FUNCTION_BLOCK Brake
VAR_INPUT
	Lh_off:BOOL;(*Left brake off signal - usually from left spring nest*)
	Lh_rubbing:BOOL; (*Left brake rubbing signal - usually from left spring nest*)
	Lh_on:BOOL; (*Left brake on signal - usually from left spring nest*)
	Lh_wear:BOOL; (*Left brake wear signal - usually from left spring nest*)
	Rh_off:BOOL; (*Right brake on signal - usually from right spring nest*)
	Rh_rubbing:BOOL; (*Right brake rubbing signal - usually from right spring nest*)
	Rh_on:BOOL; (*Right brake on signal - usually from right spring nest*)
	Rh_wear:BOOL; (*Right brake wear signal - usually from Right spring nest*)
	Lever_on:BOOL; (*Brake lever on limit switch*)
	Lever_off:BOOL; (*Brake lever off - normally from same limit switch as "Lever_on"*)
	Lever_fully_off:BOOL; (*Brake lever fully off limit switch. Necessary for automatic winders.*)
	Lh_test:BOOL; (*Left brake test switch - normally on driver's desk. Often the same switch as Lh_dump.*)
	Rh_test:BOOL; (*Right brake test switch - normally on driver's desk. Often the same switch as Rh_dump.*)
	Lh_dump:BOOL; (*Left brake dump switch - normally on driver's desk. Often the same switch as Lh_test.*)
	Rh_dump:BOOL; (*Right brake dump switch - normally on driver's desk. Often the same switch as Rh_test.*)
	Maintenance_switch:BOOL; (*Brake maintenance switch (can be on driver's desk or in control panels).*)
	Trail_brakes:BOOL; (*Trail brake control signal. Used to disable Lh_not_fully_off and Rh_not_fully_off trips.*)
	Lh_speed:INT; (*Left drum speed (normally in mm/s)*)
	Rh_speed:INT; (*Right drum speed (normally in mm/s)*)
	Movement_detect:BOOL; (*Drum movement detected (on either of the two drums in a double-drum winder)*)
	On_time:TIME; (*Maximum time allowed for brakes to apply.*)
	Off_time:TIME; (*Maximum time allowed for brakes to lift.*)
	Rubbing_speed:INT; (*Speed above which the brakes must be above the rubbing position*)
	Rubbing_time:TIME; (*Time before brake rubbing trips trigger *)
END_VAR
VAR_OUTPUT
	Maintenance:BOOL; (*The winder is in brake maintenance mode*)
	Proved_on:BOOL; (*The brake lever (if in manual mode) and both brakes are on*)
	Proved_on_500ms:BOOL; (*The brakes have been proved on for 500ms*)
	cs_Lh_off_before_rubbing:BOOL; (*The Lh_off switch has closed but the Lh_rubbing switch has not yet closed*)
	cs_Lh_on_and_rubbing:BOOL; (*The Lh_on switch has closed but the Lh_rubbing switch is still closed*)
	cs_Lh_wear_before_on:BOOL; (*The Lh_on switch has closed but the Lh_rubbing switch is still closed*)
	cs_Lh_on_and_off:BOOL; (*The Lh_on and Lh_off switches are simultaneously closed*)
	cs_Rh_off_before_rubbing:BOOL; (*The Rh_off switch has closed but the Rh_rubbing switch has not yet closed*)
	cs_Rh_on_and_rubbing:BOOL; (*The Rh_on switch has closed but the Rh_rubbing switch is still closed*)
	cs_Rh_wear_before_on:BOOL; (*The Rh_on switch has closed but the Rh_rubbing switch is still closed*)
	cs_Rh_on_and_off:BOOL; (*The Rh_on and Rh_off switches are simultaneously closed*)
	cs_Lever_off_and_on:BOOL; (*The brake lever on and off switches are simultaneously closed*)
	cs_Lever_fully_off_and_on:BOOL; (*The brake lever on and fully off switches are simultaneously closed*)
	cs_Lh_not_fully_off:BOOL; (*The brake lever has been off for longer than the brake lift time but the Lh_off switch is not closed. Trail_brakes disables this fault.*)
	cs_Rh_not_fully_off:BOOL; (*The brake lever has been off for longer than the brake lift time but the Rh_off switch is not closed. Trail_brakes disables this fault.*)
	tr_Lh_not_on:BOOL; (*The brake lever has been on for longer than the brake application time but the Lh_on switch is not closed.*)
	tr_Rh_not_on:BOOL; (*The brake lever has been on for longer than the brake application time but the Rh_on switch is not closed.*)
	tr_Lh_rubbing_trip:BOOL; (*Lh_rubbing active above the rubbing trip speed*)
	tr_Rh_rubbing_trip:BOOL; (*Rh_rubbing active above the rubbing trip speed*)
	tr_No_brake_on_in_maint:BOOL; (*The power lever was moved from the neutral position in brake maintenance mode*)
	tr_Movement_in_maint:BOOL; (*Movement has been detected in brake maintenance mode*)
	tr_Maint_switch_on:BOOL; (*The brake maintenance switch is on but a brake is not dumped*)
	hmi_Status:ARRAY[1..2] OF WORD; (*Status bits for HMI*)
END_VAR
VAR
	TON_0: TON;
	Maintenance_req: BOOL;
	RS_0: RS;
	TON_1: TON;
	TON_2: TON;
	TON_3: TON;
	TON_4: TON;
	TON_5: TON;
	TON_6: TON;
	TON_7: TON;
	TON_8: TON;
	TON_9: TON;
	TON_10: TON;
	TON_11: TON;
	TON_12: TON;
	TON_13: TON;
	TON_14: TON;
	TON_15: TON;
	TON_16: TON;
	TON_17: TON;
	BIT_TO_WORD_V0_0: BIT_TO_WORD_V0;
	BIT_TO_WORD_V0_1: BIT_TO_WORD_V0;
END_VAR

Brake_data_m();
Brake_faults();

METHOD Brake_data_m
VAR_INPUT
END_VAR
VAR
END_VAR
VAR_INST // added by the converter: edge detectors and wires of the graphical bodies
    _w1, _w2, _w3, _w4 : BOOL;
END_VAR
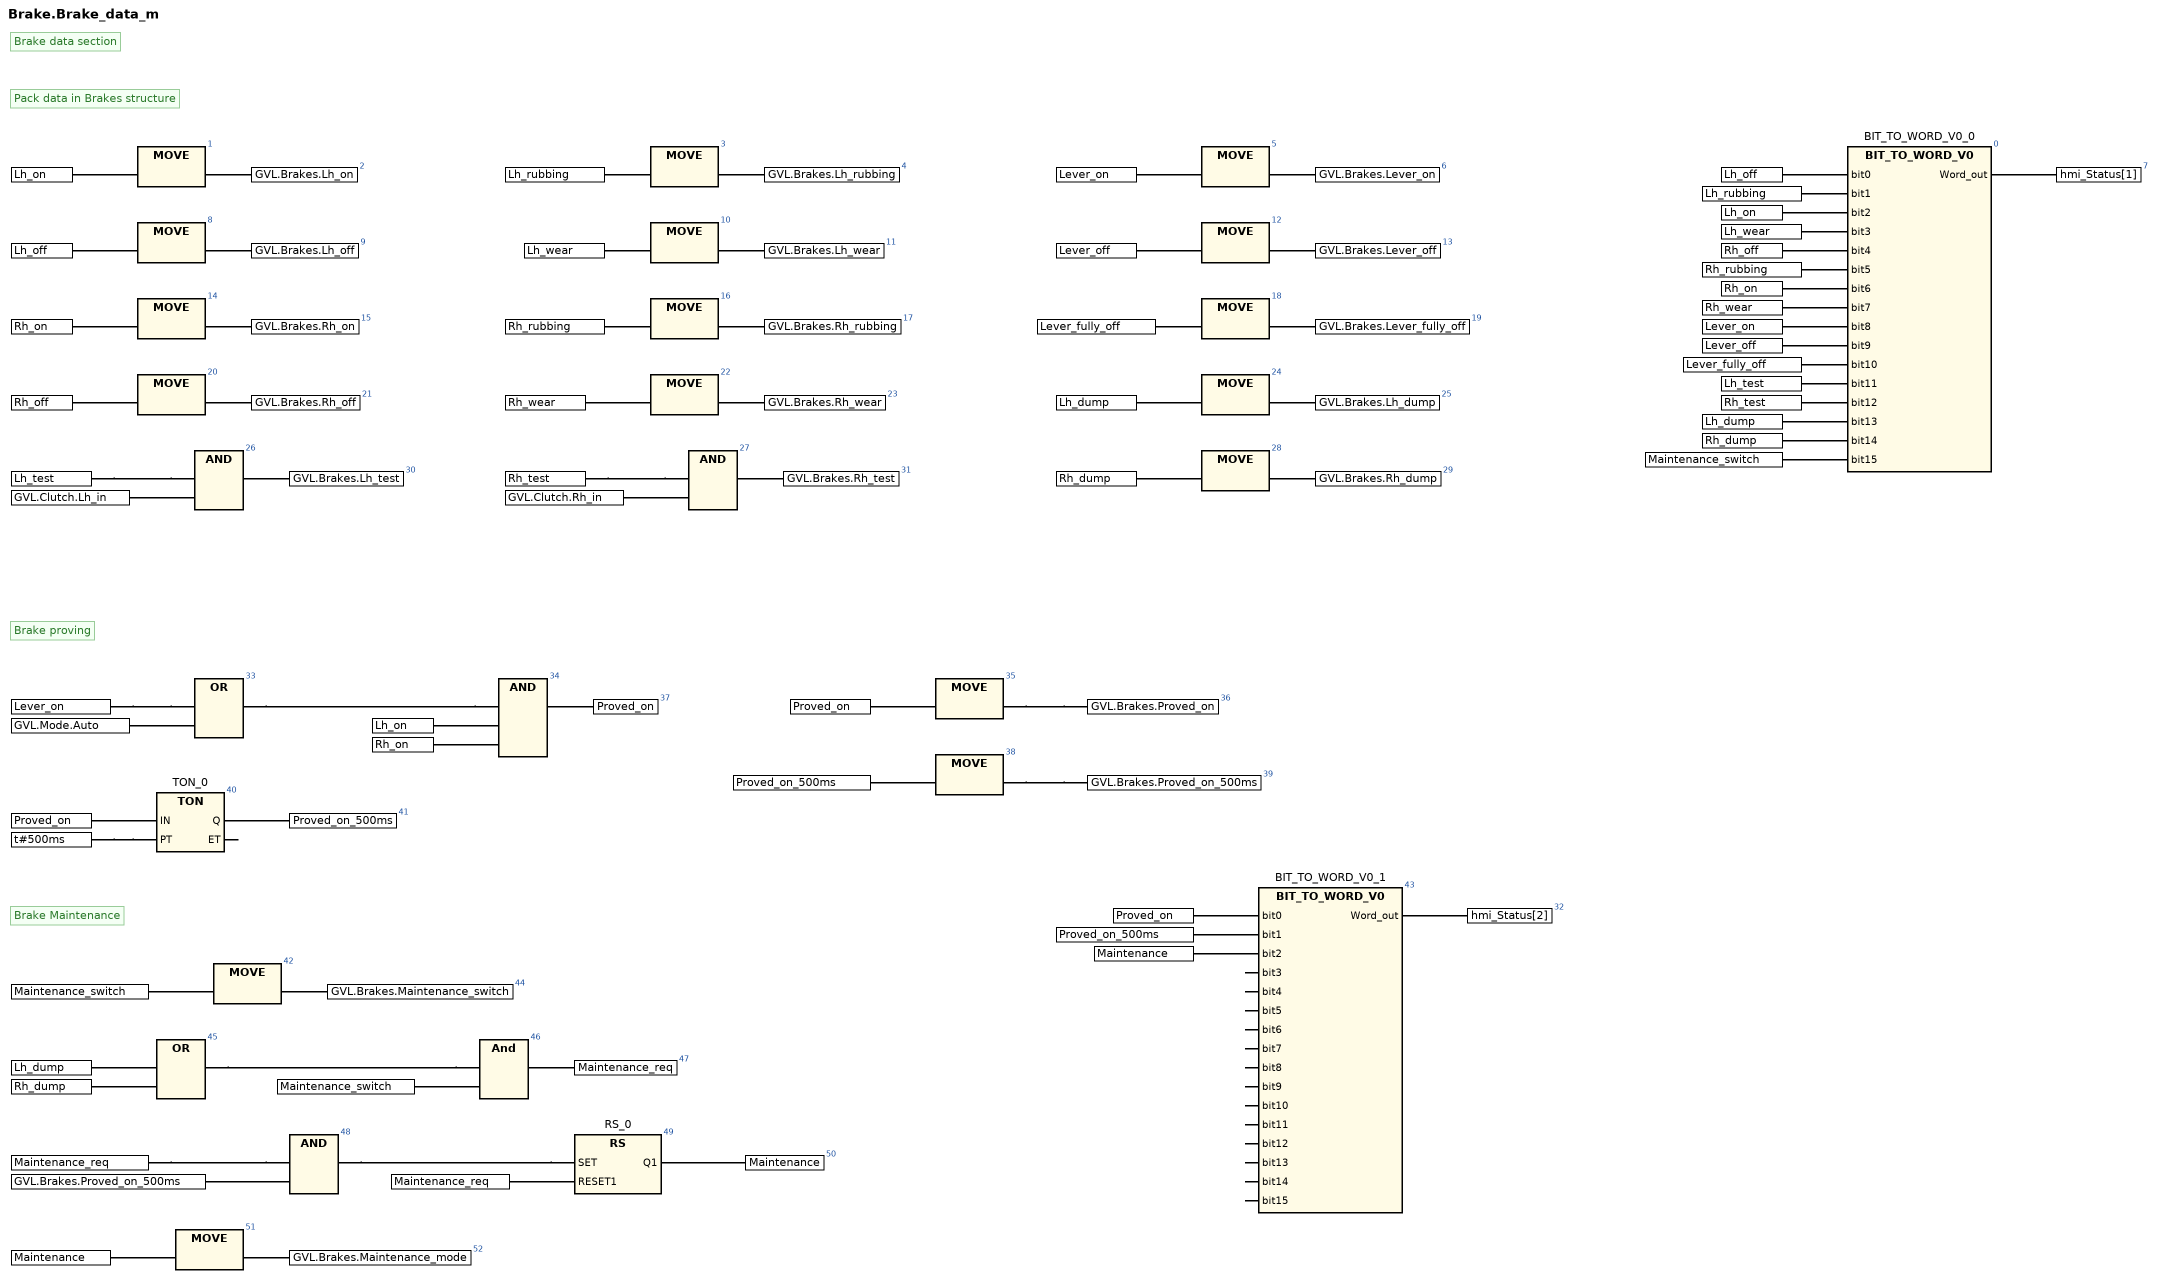
BIT_TO_WORD_V0_0(
    bit0 := Lh_off,
    bit1 := Lh_rubbing,
    bit2 := Lh_on,
    bit3 := Lh_wear,
    bit4 := Rh_off,
    bit5 := Rh_rubbing,
    bit6 := Rh_on,
    bit7 := Rh_wear,
    bit8 := Lever_on,
    bit9 := Lever_off,
    bit10 := Lever_fully_off,
    bit11 := Lh_test,
    bit12 := Rh_test,
    bit13 := Lh_dump,
    bit14 := Rh_dump,
    bit15 := Maintenance_switch); // BIT_TO_WORD_V0
// Brake data section
// Pack data in Brakes structure
GVL.Brakes.Lh_on := Lh_on;
GVL.Brakes.Lh_rubbing := Lh_rubbing;
GVL.Brakes.Lever_on := Lever_on;
hmi_Status[1] := BIT_TO_WORD_V0_0.Word_out;
GVL.Brakes.Lh_off := Lh_off;
GVL.Brakes.Lh_wear := Lh_wear;
GVL.Brakes.Lever_off := Lever_off;
GVL.Brakes.Rh_on := Rh_on;
GVL.Brakes.Rh_rubbing := Rh_rubbing;
GVL.Brakes.Lever_fully_off := Lever_fully_off;
GVL.Brakes.Rh_off := Rh_off;
GVL.Brakes.Rh_wear := Rh_wear;
GVL.Brakes.Lh_dump := Lh_dump;
_w1 := Lh_test AND GVL.Clutch.Lh_in;
_w2 := Rh_test AND GVL.Clutch.Rh_in;
GVL.Brakes.Rh_dump := Rh_dump;
GVL.Brakes.Lh_test := _w1;
GVL.Brakes.Rh_test := _w2;
hmi_Status[2] := BIT_TO_WORD_V0_1.Word_out;
// Brake proving
_w3 := (Lever_on OR GVL.Mode.Auto) AND Lh_on AND Rh_on;
GVL.Brakes.Proved_on := Proved_on;
Proved_on := _w3;
GVL.Brakes.Proved_on_500ms := Proved_on_500ms;
TON_0(IN := Proved_on, PT := t#500ms); // TON
Proved_on_500ms := TON_0.Q;
// Brake Maintenance
_w4 := Maintenance_switch;
BIT_TO_WORD_V0_1(bit0 := Proved_on, bit1 := Proved_on_500ms, bit2 := Maintenance); // BIT_TO_WORD_V0
GVL.Brakes.Maintenance_switch := _w4;
Maintenance_req := (Lh_dump OR Rh_dump) AND Maintenance_switch;
RS_0(SET := Maintenance_req AND GVL.Brakes.Proved_on_500ms, RESET1 := Maintenance_req); // RS
Maintenance := RS_0.Q1;
GVL.Brakes.Maintenance_mode := Maintenance;
END_METHOD

METHOD Brake_faults
VAR_INPUT
END_VAR
VAR_INST // added by the converter: edge detectors and wires of the graphical bodies
    _w1, _w2, _w4 : BOOL;
    _w3 : ANY;
END_VAR
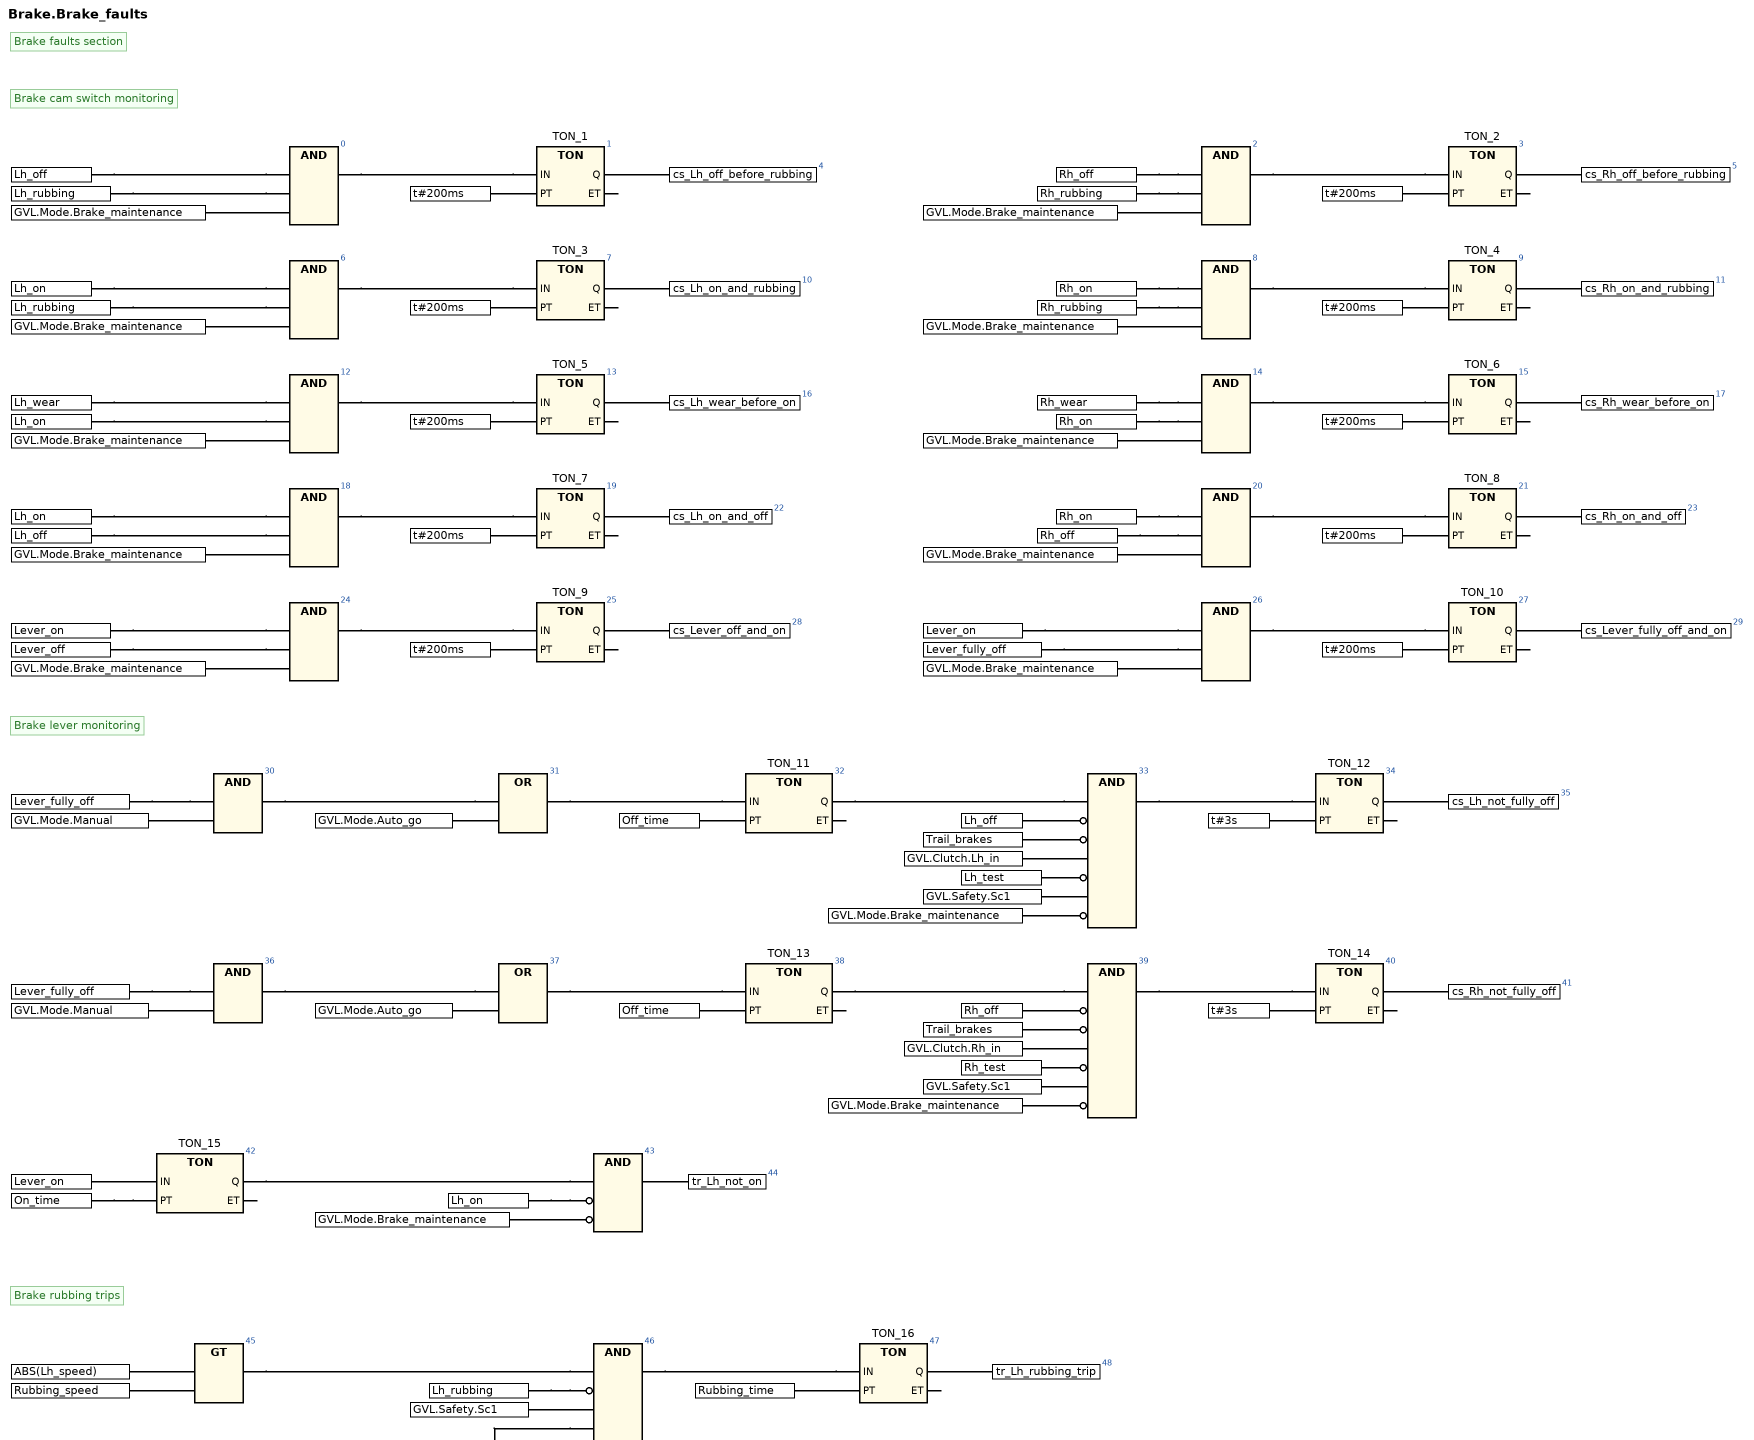
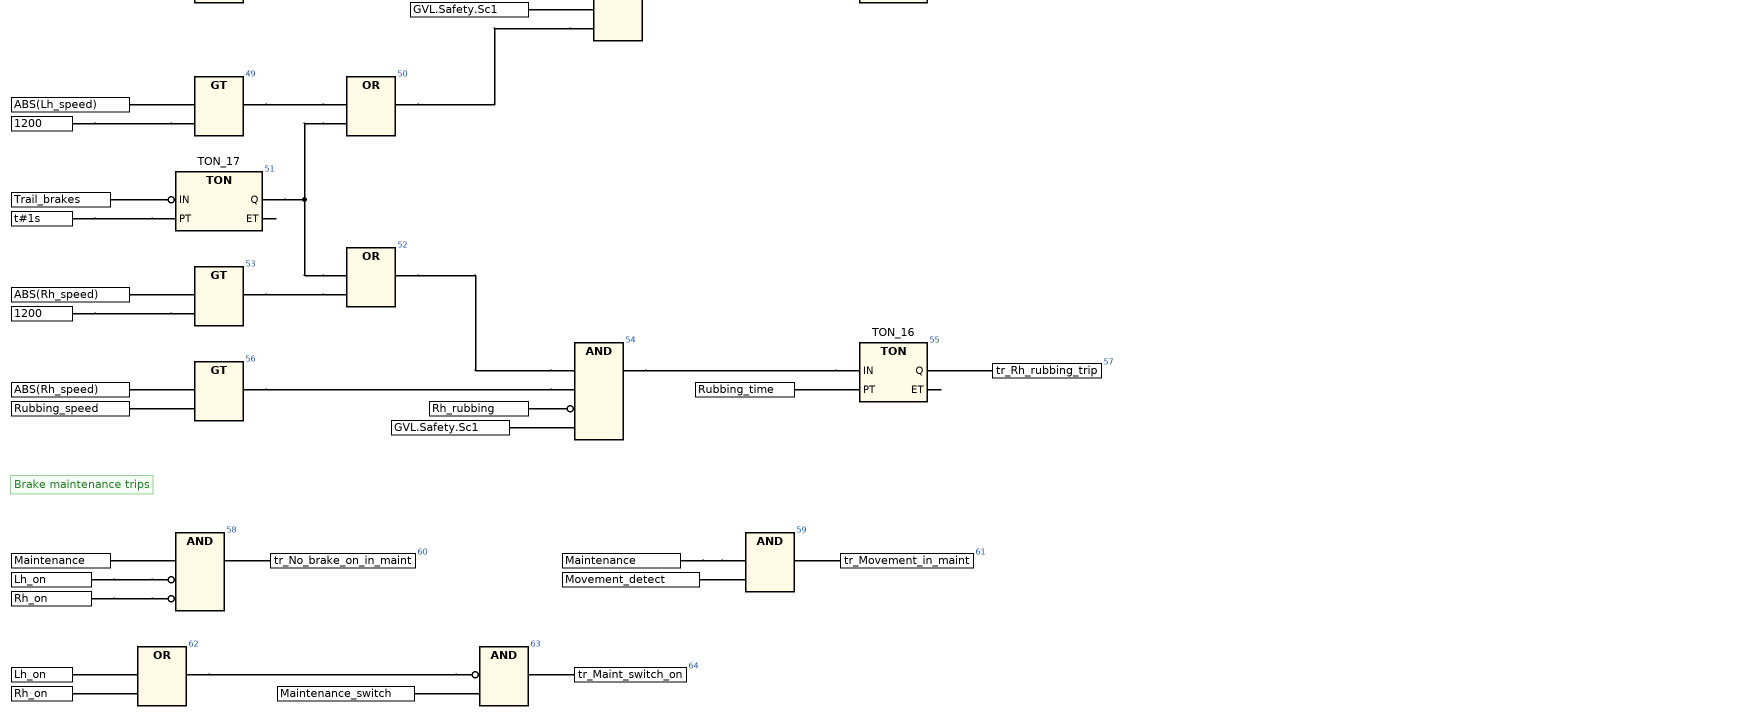
// Brake faults section
// Brake cam switch monitoring
TON_1(IN := Lh_off AND Lh_rubbing AND GVL.Mode.Brake_maintenance, PT := t#200ms); // TON
TON_2(IN := Rh_off AND Rh_rubbing AND GVL.Mode.Brake_maintenance, PT := t#200ms); // TON
cs_Lh_off_before_rubbing := TON_1.Q;
cs_Rh_off_before_rubbing := TON_2.Q;
TON_3(IN := Lh_on AND Lh_rubbing AND GVL.Mode.Brake_maintenance, PT := t#200ms); // TON
TON_4(IN := Rh_on AND Rh_rubbing AND GVL.Mode.Brake_maintenance, PT := t#200ms); // TON
cs_Lh_on_and_rubbing := TON_3.Q;
cs_Rh_on_and_rubbing := TON_4.Q;
TON_5(IN := Lh_wear AND Lh_on AND GVL.Mode.Brake_maintenance, PT := t#200ms); // TON
TON_6(IN := Rh_wear AND Rh_on AND GVL.Mode.Brake_maintenance, PT := t#200ms); // TON
cs_Lh_wear_before_on := TON_5.Q;
cs_Rh_wear_before_on := TON_6.Q;
TON_7(IN := Lh_on AND Lh_off AND GVL.Mode.Brake_maintenance, PT := t#200ms); // TON
TON_8(IN := Rh_on AND Rh_off AND GVL.Mode.Brake_maintenance, PT := t#200ms); // TON
cs_Lh_on_and_off := TON_7.Q;
cs_Rh_on_and_off := TON_8.Q;
TON_9(IN := Lever_on AND Lever_off AND GVL.Mode.Brake_maintenance, PT := t#200ms); // TON
TON_10(IN := Lever_on AND Lever_fully_off AND GVL.Mode.Brake_maintenance, PT := t#200ms); // TON
cs_Lever_off_and_on := TON_9.Q;
cs_Lever_fully_off_and_on := TON_10.Q;
// Brake lever monitoring
TON_11(IN := Lever_fully_off AND GVL.Mode.Manual OR GVL.Mode.Auto_go, PT := Off_time); // TON
TON_12(IN := TON_11.Q AND NOT Lh_off AND NOT Trail_brakes AND GVL.Clutch.Lh_in AND NOT Lh_test AND GVL.Safety.Sc1 AND NOT GVL.Mode.Brake_maintenance, PT := t#3s); // TON
cs_Lh_not_fully_off := TON_12.Q;
TON_13(IN := Lever_fully_off AND GVL.Mode.Manual OR GVL.Mode.Auto_go, PT := Off_time); // TON
TON_14(IN := TON_13.Q AND NOT Rh_off AND NOT Trail_brakes AND GVL.Clutch.Rh_in AND NOT Rh_test AND GVL.Safety.Sc1 AND NOT GVL.Mode.Brake_maintenance, PT := t#3s); // TON
cs_Rh_not_fully_off := TON_14.Q;
TON_15(IN := Lever_on, PT := On_time); // TON
tr_Lh_not_on := TON_15.Q AND NOT Lh_on AND NOT GVL.Mode.Brake_maintenance;
// Brake rubbing trips
TON_16(IN := (ABS(Lh_speed)) > Rubbing_speed AND NOT Lh_rubbing AND GVL.Safety.Sc1 AND _w1, PT := Rubbing_time); // TON
tr_Lh_rubbing_trip := TON_16.Q;
_w1 := (ABS(Lh_speed)) > 1200 OR TON_17.Q;
TON_17(IN := NOT Trail_brakes, PT := t#1s); // TON
_w3 := TON_17.Q OR _w2;
_w2 := (ABS(Rh_speed)) > 1200;
TON_16(IN := _w3 AND _w4 AND NOT Rh_rubbing AND GVL.Safety.Sc1, PT := Rubbing_time); // TON
_w4 := (ABS(Rh_speed)) > Rubbing_speed;
tr_Rh_rubbing_trip := TON_16.Q;
// Brake maintenance trips
tr_No_brake_on_in_maint := Maintenance AND NOT Lh_on AND NOT Rh_on;
tr_Movement_in_maint := Maintenance AND Movement_detect;
tr_Maint_switch_on := NOT (Lh_on OR Rh_on) AND Maintenance_switch;
END_METHOD

END_FUNCTION_BLOCK

(* stored: Version 1.1.0.1, ProductVersion 3.1.4024.0
   POU Brake: Id {8299c612-9708-4d8b-9a02-4771041e89b7}, SpecialFunc None
   Method Brake_data_m: Id {b01e94a7-ee2d-4698-b277-739dbefaaf40}
   Method Brake_faults: Id {6af2cde8-de97-41bc-9d52-dd2ca2e2c179} *)
